(*
SPDX-FileCopyrightText: © 2026 Oleksandr Tiutyk <trofimich@gmail.com>
SPDX-License-Identifier: MIT
License: https://opensource.org/license/mit
*)

(*!
<summary>Performs a cyclic file byte transfer through a borrowed file resource.</summary>
<description>
Configure SourceBuffer and BytesCountToWrite before Start and keep them stable until STOPPED. The caller owns
the buffer and must keep at least the requested number of bytes readable and unchanged through stopping. A
null buffer or zero count raises DataMemberNotSpecifiedException before the native request; the base Task
records FAILURE and completes its cleanup. Buffer capacity and the validity of non-null addresses are caller
preconditions, not checked here. No ownership is transferred and partial I/O effects are not rolled back.
</description>
*)

{attribute 'no_explicit_call' := 'do not call this function block directly'}
FUNCTION_BLOCK WriteBytesToFile EXTENDS FileContentTask
VAR_STAT
	//! <summary>Static type metadata available before the base task initializes its default name.</summary>
	{attribute 'hide'}
	_ClassName : STRING := __POUNAME();
END_VAR
VAR
    _WriteBytes : Tc2_System.FB_FileWrite;
END_VAR

(*!
<summary>Reports the byte count from a successfully completed write.</summary>
<description>
Returns the native result only while State.Stopped and FinalStopReason.WorkDone are both TRUE. In every other
state, including READY, RUNNING, failure and cancellation, returns the initial value of the property type.
This default is not a success indicator; inspect the task state and final reason. Zero after failure or
cancellation does not mean no bytes were written; partial native effects are not rolled back. The getter does
not modify native outputs or buffers. Copy a successful result before Reset or reuse.
</description>
*)
{attribute 'monitoring' := 'call'}
PROPERTY ActuallyWrittenBytes : UDINT
GET
IF NOT State.Stopped OR_ELSE NOT FinalStopReason.WorkDone THEN
	RETURN;
END_IF

ActuallyWrittenBytes := _WriteBytes.cbWrite;
END_GET
END_PROPERTY

(*!
<summary>Exposes the native operation target copied from the bound file resource.</summary>
<description>
The resource target overwrites a separately assigned value before native submission. Configure the resource
owner to select a target; do not change this value while the task is running.
</description>
*)
{attribute 'monitoring' := 'call'}
PROPERTY AmsNetId : Tc2_System.T_AmsNetID
GET
AmsNetId := _WriteBytes.sNetId;
END_GET
SET
_WriteBytes.sNetId := AmsNetId;
END_SET
END_PROPERTY

(*!
<summary>Specifies the requested byte count.</summary>
<description>
Must be positive and no greater than the available buffer capacity. Zero is rejected by OnRunning before the
native request and results in Task FAILURE after cleanup. The setter stores configuration without validation;
keep the count stable from Start until STOPPED.
</description>
*)
{attribute 'monitoring' := 'call'}
PROPERTY BytesCountToWrite : UDINT
GET
BytesCountToWrite := _WriteBytes.cbWriteLen;
END_GET
SET
_WriteBytes.cbWriteLen := BytesCountToWrite;
END_SET
END_PROPERTY

(*!
<summary>Provides the concrete type name used in diagnostics.</summary>
<description>
Returns borrowed read-only metadata; keep the instance alive and do not modify the referenced string.
Initialized static storage is ready during base Task.FB_init; this getter has no side effects or exceptions.
</description>
*)
{attribute 'monitoring' := 'call'}
PROPERTY ClassName : REFERENCE TO STRING
GET
ClassName REF= _ClassName;
END_GET
END_PROPERTY

(*!
<summary>Reports whether the underlying native file operation is busy.</summary>
<description>
Observes native I/O, including work drained during stopping. FALSE is not a task-success result and does not
independently permit the resource owner to close or destroy the file.
</description>
*)
{attribute 'monitoring' := 'call'}
PROPERTY FileOperationInProgress : BOOL
GET
FileOperationInProgress := _WriteBytes.bBusy;
END_GET
END_PROPERTY

(*!
<summary>Provides the library namespace used in diagnostics.</summary>
<description>Returns borrowed read-only namespace storage; do not modify the referenced string.</description>
*)
{attribute 'monitoring' := 'call'}
PROPERTY NamespaceName : REFERENCE TO STRING
GET
NamespaceName REF= CurrentNamespace.Name;
END_GET
END_PROPERTY

(*!
<summary>Resets the native request edge after the task has stopped.</summary>
<description>
Also preserves the inherited resource-binding cleanup. Configured inputs remain available for reuse; borrowed
buffers are not freed or cleared. Pending I/O must finish during stopping before this hook runs.
</description>
*)
METHOD PROTECTED OnReset
SUPER^.OnReset();

_WriteBytes(bExecute := FALSE);
END_METHOD

(*!
<summary>Writes the configured byte buffer to the bound file and checks the written count.</summary>
<description>
Requires a live bound resource whose owner keeps the handle acquired until stopping completes. Before
submitting I/O, a null buffer or zero count raises DataMemberNotSpecifiedException for the missing property.
This rejects invalid configuration through the base Task failure and cleanup path. Native errors also raise an
exception without dynamic string-builder allocations; completed I/O effects are not rolled back.
</description>
<param name="processingState">BUSY while pending; DONE after a full write; ERROR on a short write.</param>
<param name="stopReasonMessage">
Receives byte-count diagnostics on a short write; native failures use exceptions.
</param>
*)
METHOD PROTECTED OnRunning
VAR_OUTPUT
	processingState : TOF_Tasks.TASK_PROCESSING_STATE;
END_VAR
VAR_IN_OUT
	stopReasonMessage : TOF_Core.ERROR_MESSAGE;
END_VAR
VAR
	errorMessage : TOF_Core.ERROR_MESSAGE;
END_VAR
IF NOT _WriteBytes.bExecute THEN 
	IF NOT __ISVALIDREF(_FileHandleResource) THEN
		TOF_Core.Exceptions.ThrowDataMemberNotSpecified(
			sourceNamespaceName := NamespaceName,
			sourceClassName := ClassName,
			sourcePOUName := __POUNAME(),
			sourcePosition := __POSITION(),
			dataMemberName := 'FileHandleResource'
		);		
	END_IF
	
	IF _WriteBytes.pWriteBuff = TOF_Core.Memory.NULL_ADDRESS THEN
		TOF_Core.Exceptions.ThrowDataMemberNotSpecified(
			sourceNamespaceName := NamespaceName,
			sourceClassName := ClassName,
			sourcePOUName := __POUNAME(),
			sourcePosition := __POSITION(),
			dataMemberName := 'SourceBuffer'
		);
	END_IF

	IF _WriteBytes.cbWriteLen = TOF_Core.UnsignedInt32.ZERO THEN
		TOF_Core.Exceptions.ThrowDataMemberNotSpecified(
			sourceNamespaceName := NamespaceName,
			sourceClassName := ClassName,
			sourcePOUName := __POUNAME(),
			sourcePosition := __POSITION(),
			dataMemberName := 'BytesCountToWrite'
		);
	END_IF

	_WriteBytes.sNetId := _FileHandleResource.AmsNetId;
	_WriteBytes.hFile := _FileHandleResource.FileHandle;
END_IF

_WriteBytes(bExecute := TRUE);

IF _WriteBytes.bError THEN
	TOF_Core.WideStrings.Append255(
		errorMessage,
		"An error occurred while writing bytes to file ",
		TO_WSTRING(FilePath),
		"'");

	FileSystemExceptions.ThrowFileSystem(
		sourceNamespaceName := NamespaceName,
		sourceClassName := ClassName,
		sourcePOUName := __POUNAME(),
		sourcePosition := __POSITION(),
		message := errorMessage,
		errorCode := _WriteBytes.nErrId
	);
END_IF

IF NOT _WriteBytes.bBusy THEN
	(* A short write may leave bError=FALSE; success requires the full byte count. *)
	IF _WriteBytes.cbWrite <> _WriteBytes.cbWriteLen THEN
		stopReasonMessage := TOF_Core.WideStrings.Concat255(
			"File write byte count mismatch: expected ",
			TO_WSTRING(_WriteBytes.cbWriteLen),
			", written ",
			TO_WSTRING(_WriteBytes.cbWrite)
		);
		
		processingState := TOF_Tasks.TASK_PROCESSING_STATE.ERROR;
	ELSE
		processingState := TOF_Tasks.TASK_PROCESSING_STATE.DONE;
	END_IF
END_IF
END_METHOD

(*!
<summary>Wait for an already submitted file operation before allowing handle release.</summary>
<description>
FALSE on bExecute only avoids a new request; it does not abort the pending one. Runs for every stop reason. If
no operation is busy, stopping is ready immediately.
</description>
<param name="readyToRelease">TRUE after pending work has completed and release may begin.</param>
*)

METHOD PROTECTED OnStopping
VAR_OUTPUT
	readyToRelease : BOOL;
END_VAR
IF _WriteBytes.bBusy THEN
	_WriteBytes(bExecute := FALSE);
END_IF

readyToRelease := NOT _WriteBytes.bBusy;
END_METHOD

(*!
<summary>Reports the size of this concrete instance in bytes.</summary>
*)
{attribute 'monitoring' := 'call'}
PROPERTY SelfSize : ULINT
GET
SelfSize := XSIZEOF(THIS^);
END_GET
END_PROPERTY

(*!
<summary>Provides the caller-owned buffer address for the transfer.</summary>
<description>
Must be non-null before I/O. The caller provides at least BytesCountToWrite bytes of readable and unchanged
storage and retains it until STOPPED, including cancellation cleanup. The setter stores the address without
validating capacity or lifetime; a null address is rejected by OnRunning before the native request. Keep this
setting stable during the run.
</description>
*)
{attribute 'monitoring' := 'call'}
PROPERTY SourceBuffer : PVOID
GET
SourceBuffer := _WriteBytes.pWriteBuff;
END_GET
SET
_WriteBytes.pWriteBuff := SourceBuffer;
END_SET
END_PROPERTY

(*!
<summary>Configures the timeout passed to native operation requests.</summary>
<description>
Set before Start and keep unchanged until STOPPED. Reset preserves this value. It is not an overall task
deadline or a guarantee of resource release after a timeout.
</description>
*)
{attribute 'monitoring' := 'call'}
PROPERTY Timeout : TIME
GET
Timeout := _WriteBytes.tTimeout;
END_GET
SET
_WriteBytes.tTimeout := Timeout;
END_SET
END_PROPERTY

END_FUNCTION_BLOCK

(* stored: Version 1.1.0.1
   POU WriteBytesToFile: Id {7fb15e59-abf9-416d-bf95-7588c3be0b84}, SpecialFunc None
   Folder Inputs: Id {8897b775-17bd-40ce-8805-3927b593ee47}
   Folder Outputs: Id {4376422b-0adc-434a-b1d5-87c1f2710313}
   Folder Overriden methods: Id {d0605ba9-7e66-4361-bc98-1fe639a51c56}
   Property ActuallyWrittenBytes: Id {197d4ba0-9df3-4f5f-b648-e57b58220522}
   Get Get: Id {242ce73c-3465-4c93-a5ea-fbdaf2402c04}
   Property AmsNetId: Id {a24a2093-593c-4aaf-b5ce-1c5dbc3b4755}
   Get Get: Id {40e747b3-ef49-4ade-aaa2-5e2addcefd5c}
   Set Set: Id {99591f2a-a541-4d55-a6d0-2ddb6c10dc9d}
   Property BytesCountToWrite: Id {df3b5887-8f47-4a2e-a3de-11d5df1acd6d}
   Get Get: Id {2a2b0e76-fb84-4085-b06b-ce8fd99a0749}
   Set Set: Id {7f86b8d4-754a-4624-b8ba-ad18ccb44893}
   Property ClassName: Id {292b66ee-18c0-4078-befa-5ba54f7cb1aa}
   Get Get: Id {3fd7ed9c-f859-42d5-9dd7-80edfc25c3a6}
   Property FileOperationInProgress: Id {dec96700-4c27-4085-b567-037497945de8}
   Get Get: Id {9a19ffab-a886-4858-85ae-7700db207ea7}
   Property NamespaceName: Id {46067b07-021a-4c1d-928e-c925a93bb725}
   Get Get: Id {9b9db4ed-afad-48d6-b776-2729cf166199}
   Method OnReset: Id {2a0ac1a8-8e3d-47b4-8633-8e7e44e211d7}
   Method OnRunning: Id {1441cdc8-acfb-4842-a5f8-6dffac4135e4}
   Method OnStopping: Id {0e54eed8-3851-4bfb-8d95-75b4cf2d9c12}
   Property SelfSize: Id {f485ccb4-946c-4324-9dd2-3933e7d9c49f}
   Get Get: Id {49a23a78-3b91-48aa-b262-eed842537e31}
   Property SourceBuffer: Id {9a130528-f270-44f7-9c13-ad3099c5d067}
   Get Get: Id {6bbe71f9-f6bb-4d14-a6f7-3f57edb989b5}
   Set Set: Id {83450a3e-1930-420f-9c4d-7ec75e9da792}
   Property Timeout: Id {2787d246-759b-4387-947c-e77d36299545}
   Get Get: Id {d6e1717c-c8b8-446d-a044-e9c2a53fb28b}
   Set Set: Id {f862d09e-641d-4fe1-bbe1-065a84b5d885} *)
